{attribute 'monitoring':='call'}
INTERFACE I_CameraSink

METHOD AddCamPoint : BOOL
VAR_INPUT
	sDeformationPoint	: ST_DeformationPointAccurate;
END_VAR
END_METHOD

METHOD AddTeachPoint : BOOL
VAR_INPUT
  sTeachPoint : ST_DeformationPointAccurate;
END_VAR
END_METHOD

(*
  Event cam done "detecting points", sheet/repeate done.
  Called after last point will be streamed to same CT.
*)
METHOD CamDone : BOOL
END_METHOD

(*
  Event cam started "detecting points".
  Is called before streaming cam points.
*)
METHOD CamStarted
VAR_INPUT
  nX0 : DINT; // detected start position
END_VAR
END_METHOD

// Detected "real" image lenght [m]
PROPERTY fPrintLengthEffective : LREAL
SET
END_SET
END_PROPERTY

END_INTERFACE

(* stored: Version 1.1.0.1, ProductVersion 3.1.4024.11
   Itf I_CameraSink: Id {c7f13400-6272-4109-9d42-da2a605cebc8}
   Method AddCamPoint: Id {8c397612-ef52-42b0-92b4-df25225c5d90}
   Method AddTeachPoint: Id {01dedd52-bc68-4f3e-b5ba-be065d82bed2}
   Method CamDone: Id {dae457a0-f1b8-4ae1-bdb6-7fab81b30ff7}
   Method CamStarted: Id {6167fba8-5e99-4ef2-8c53-3654b01163aa}
   Property fPrintLengthEffective: Id {5d63e249-80f2-46a4-99a2-53ffff682b1b}
   Set Set: Id {cf186f9b-7da7-4af1-ab5c-0f79c1576da9} *)
